{attribute 'enable_dynamic_creation'}
FUNCTION_BLOCK FB_Needle EXTENDS FB_UsingPiece
VAR_INPUT
END_VAR
VAR_OUTPUT
END_VAR
VAR
	pSeptum : POINTER TO FB_PieceBase;
END_VAR

METHOD FB_init : BOOL
VAR_INPUT
	bInitRetains : BOOL; // if TRUE, the retain variables are initialized (warm start / cold start)
	bInCopyCode : BOOL;  // if TRUE, the instance afterwards gets moved into the copy code (online change)
END_VAR
bUsingPiece := TRUE;
eObjectType := E_ObjectType.OBJECTTYPE_Needle;
eObjectGroup := E_ObjectGroup.OBJECTGROUP_Piece;
END_METHOD

{attribute 'object_name' := 'M_ClearAllProps'}
METHOD M_ClearAllProps

VAR_INPUT
	bIgnoreParent : BOOL; //Es wird das gesamte OD gelöscht. -> Zeiger auf Parent nicht mehr gültig!
END_VAR
pSeptum := 0;
SUPER^.M_ClearAllProps(bIgnoreParent);
END_METHOD

PROPERTY P_pLatestChild : POINTER TO FB_PieceBase
GET
IF pSeptum > 0 THEN
	P_pLatestChild := pSeptum;	
ELSE
	P_pLatestChild := THIS;
END_IF
END_GET
END_PROPERTY

PROPERTY P_pSeptum : POINTER TO FB_PieceBase
GET
P_pSeptum := pSeptum;
END_GET
SET
pSeptum := P_pSeptum;
END_SET
END_PROPERTY

END_FUNCTION_BLOCK

(* stored: Version 1.1.0.1, ProductVersion 3.1.4022.18
   POU FB_Needle: Id {b2034c4d-1a23-40c9-bc9e-1e65b2b4ec40}, SpecialFunc None
   Method FB_init: Id {72005d1a-7382-4bf3-9d4e-aa8ef066ce21}
   Method M_ClearAllProps: Id {c3c96786-53ab-4e3f-ad24-7a2851f05848}
   Property P_pLatestChild: Id {c328820f-c8a6-4393-b477-1988fb97d247}
   Get Get: Id {2be5f538-681b-4b65-b198-ab07c7bdd706}
   Property P_pSeptum: Id {0c977316-4644-4bec-9869-8076a1584c71}
   Get Get: Id {e6b0c0ee-a929-4d6d-8126-a548d67cd7f7}
   Set Set: Id {da306de2-81a3-42a9-b548-cf0db607ac2b} *)
